FUNCTION_BLOCK UXIntComparer EXTENDS Object IMPLEMENTS IComparer
VAR
	_ClassName : STRING := __POUNAME();
END_VAR

{attribute 'monitoring' := 'call'}
PROPERTY ClassName : STRING
GET
ClassName := _ClassName;
END_GET
END_PROPERTY

{attribute "object_name" := "Compare"}
METHOD Compare : COMPARISION_RESULT
VAR_INPUT
	left : PVOID;
	right : PVOID;
END_VAR
VAR
	leftPointer : POINTER TO __UXINT; 
	rightPointer : POINTER TO __UXINT; 
END_VAR
IF left = 0 AND right = 0 THEN
	Compare := COMPARISION_RESULT.EQUALS;
	RETURN;
END_IF

IF left = 0 THEN
	Compare := COMPARISION_RESULT.LEFT_LESS_RIGHT;
	RETURN;	
END_IF

IF right = 0 THEN
	Compare := COMPARISION_RESULT.LEFT_GREATER_RIGHT;
	RETURN;	
END_IF

leftPointer := left;
rightPointer := right;

IF leftPointer^ < rightPointer^ THEN
	Compare := COMPARISION_RESULT.LEFT_LESS_RIGHT;
ELSIF leftPointer^ > rightPointer^ THEN
	Compare := COMPARISION_RESULT.LEFT_GREATER_RIGHT;
ELSE
	Compare := COMPARISION_RESULT.EQUALS;	
END_IF
END_METHOD

END_FUNCTION_BLOCK

(* stored: Version 1.1.0.1
   POU UXIntComparer: Id {46b094cf-0d83-43dd-8f55-8c90ddd9417a}, SpecialFunc None
   Property ClassName: Id {3d1e4338-d3e6-497c-97d6-0ac58f71bef5}
   Get Get: Id {db0bdfc1-7f8e-41fc-95ee-bc780c15b1fb}
   Method Compare: Id {498c52ad-f6a6-4d11-bc99-94b2aae0c28f} *)
